// TIA Portal V20 export
TYPE "LKinCtrl_typePnPParameter"
   STRUCT
      direction : Array[1..3] of LReal;   // Direction of vector (will be normed by FB) from start / target
      workingHeight : LReal := 0.0;   // Length of vector
      transitionArea : LReal := 0.0;   // Permissible blending area at end of vector
      dynamicsFactor : LReal := 100.0;   // Path dynamics scaling factor
   END_STRUCT;
END_TYPE
